# B&R Automation Studio project testing1
Automation Studio 4.6.3.55 SP

## Configuration Config1

### Task classes (Cpu.sw)
```
Cyclic#4:
  Program <- Program.prg
  Program1 <- Program1.prg
```

### Hardware
```
X20CP1586 : X20CP1586 v1.5.0.0
  Connector IF2:
    ActivateDevice = 1
  ConfigurationID = testing1_Config1
  Simulation = 1
```

## Logical view

- Visualisation Logical/mappView (not shown)

### Program Logical/Program (IEC)

#### Init.st
```iecst
PROGRAM _INIT
	Speed := 30;
	Temperature := 20;

END_PROGRAM
```

Listed in the project but not available here: Logical/Global.typ, Logical/Global.var, Logical/Libraries, Logical/Program1
